(* PLC project SafeLOGIC, BrAutomation SafeDESIGNER  5.24.1.0 *)
(* stored: companyURL http://www.br-automation.com, creationDateTime Thu Sep 25 11:19:38 2025 *)

PROGRAM HW_MIN_MON
  VAR  (* added by the conversion: wires and edge detectors of the diagram *)
    _NOT_S36_OUT : ANY;
  END_VAR

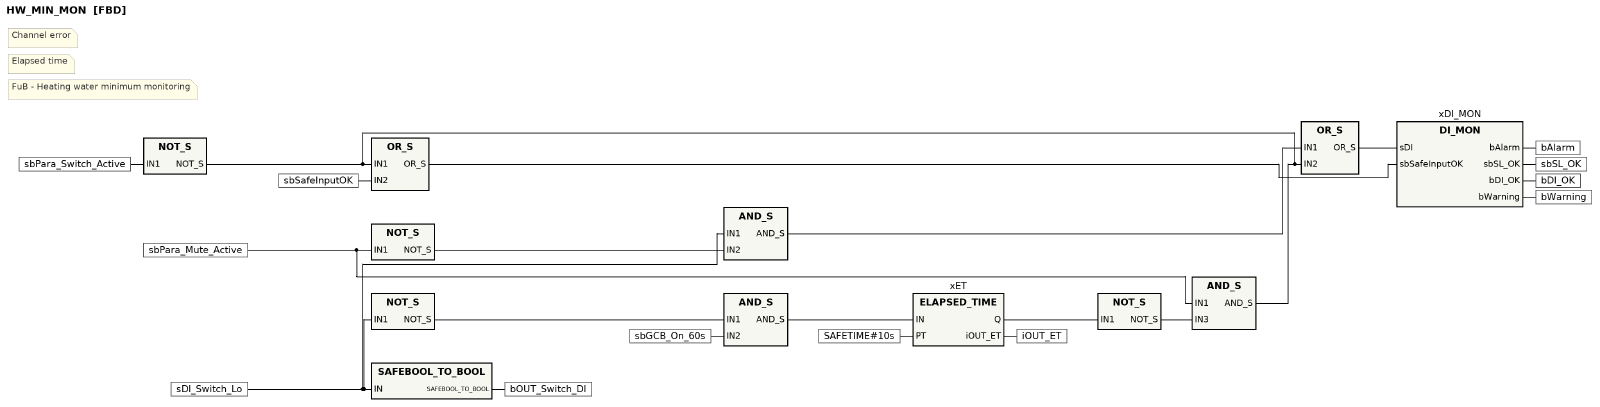
(* FBD diagram, written out as Structured Text *)
(* FuB - Heating water minimum monitoring *)
bOUT_Switch_DI := SAFEBOOL_TO_BOOL(sDI_Switch_Lo);
xET(IN := AND_S(NOT_S(sDI_Switch_Lo), sbGCB_On_60s), PT := SAFETIME#10s);
_NOT_S36_OUT := NOT_S(sbPara_Switch_Active);
xDI_MON(sDI := OR_S(AND_S(sDI_Switch_Lo, NOT_S(sbPara_Mute_Active)), AND_S(sbPara_Mute_Active, NOT_S(xET.Q)), _NOT_S36_OUT), sbSafeInputOK := OR_S(_NOT_S36_OUT, sbSafeInputOK));
bAlarm := xDI_MON.bAlarm;
(* Elapsed time *)
iOUT_ET := xET.iOUT_ET;
bDI_OK := xDI_MON.bDI_OK;
sbSL_OK := xDI_MON.sbSL_OK;
(* Channel error *)
bWarning := xDI_MON.bWarning;
END_PROGRAM
